(* IEC 61131-3 sources: repolevel_ST_code_completion/output/full_case_fixed/repoeval_elevator/readful_result, 5 files *)

(* ---- F_DetectCurrentFloor.st ---- *)
FUNCTION F_DetectCurrentFloor : INT
VAR_INPUT
FloorSensor0	:	BOOL;		// 0楼传感器
FloorSensor1	:	BOOL;		// 1楼传感器
FloorSensor2	:	BOOL;		// 2楼传感器
FloorSensor3	:	BOOL;		// 3楼传感器
CurrentFloor	:	INT;		// 当前楼层（用于保持状态）
END_VAR
IF FloorSensor0 THEN
F_DetectCurrentFloor := 0;
ELSIF FloorSensor1 THEN
F_DetectCurrentFloor := 1;
ELSIF FloorSensor2 THEN
F_DetectCurrentFloor := 2;
ELSIF FloorSensor3 THEN
F_DetectCurrentFloor := 3;
ELSE
F_DetectCurrentFloor := 0; // Default valid floor value if no sensors are active
END_IF;
RETURN;
END_FUNCTION

(* ---- F_RegisterCalls.st ---- *)
FUNCTION F_RegisterCalls
VAR_INPUT
 CallGround		:	BOOL;		// 0楼呼叫
 CallFloor1		:	BOOL;		// 1楼呼叫
 CallFloor2		:	BOOL;		// 2楼呼叫
 CallFloor3		:	BOOL;		// 3楼呼叫
END_VAR
VAR_IN_OUT
 TargetFloors	:	ARRAY[0..3] OF BOOL;	// 目标楼层数组
END_VAR
IF CallGround THEN
 TargetFloors[0] := TRUE;
END_IF

IF CallFloor1 THEN
 TargetFloors[1] := TRUE;
END_IF

IF CallFloor2 THEN
 TargetFloors[2] := TRUE;
END_IF

IF CallFloor3 THEN
 TargetFloors[3] := TRUE;
END_IF

RETURN;
END_FUNCTION

(* ---- F_UpdateDoorAnimation.st ---- *)
FUNCTION F_UpdateDoorAnimation : DINT
VAR_INPUT
bOpenDoor		:	BOOL;		// 开门命令
bCloseDoor		:	BOOL;		// 关门命令
bCallFloor		:	BOOL;		// 该楼层有呼叫
nCurrentAni		:	DINT;		// 当前动画值
nMaxAni			:	DINT := 70;	// 最大动画值
END_VAR
VAR
nNewAni			:	DINT;		// 新的动画值
END_VAR

nNewAni := nCurrentAni;

// 开门动画（增加动画值）
IF bOpenDoor AND nNewAni < nMaxAni AND bCallFloor THEN
nNewAni := nNewAni + 1;
END_IF

// 关门动画（减少动画值）
IF bCloseDoor AND nNewAni > 0 THEN
nNewAni := nNewAni - 1;
END_IF

F_UpdateDoorAnimation := nNewAni;
END_FUNCTION

(* ---- FB_ElevatorDoorController.st ---- *)
FUNCTION_BLOCK FB_ElevatorDoorController
VAR_INPUT
	bArrivedAtTarget	:	BOOL;		// 到达目标楼层
	bDoorClosed			:	BOOL;		// 门已关闭传感器
END_VAR
VAR_OUTPUT
	bOpenDoor			:	BOOL;		// 开门命令
	bCloseDoor			:	BOOL;		// 关门命令
	bDoorOpen			:	BOOL;		// 门打开状态
	bDoorReady			:	BOOL;		// 门准备好（可以移动）
END_VAR
VAR
	fbDoorTimer			:	TON;		// 开门延时定时器
	fbCloseDoorTimer	:	TON;		// 关门延时定时器
	nState				:	INT;		// 状态机
END_VAR

CASE nState OF
	0: // 空闲状态
		bOpenDoor := FALSE;
		bCloseDoor := FALSE;
		bDoorReady := TRUE;

		IF bArrivedAtTarget THEN
			nState := 1; // 开始开门流程
		END_IF

1: // 开门延时
    bCloseDoor := FALSE;
    bDoorReady := FALSE;
    fbDoorTimer.IN := TRUE;
    fbDoorTimer.PT := T#2S;

    IF fbDoorTimer.Q THEN
      fbDoorTimer.IN := FALSE;
      nState := 2; // 开门命令
    END_IF

	2: // 开门命令
		bOpenDoor := TRUE;
		bDoorOpen := TRUE;
		bDoorReady := FALSE;

		IF NOT bArrivedAtTarget THEN
			nState := 3; // 开始关门流程
		END_IF

3: // 关门延时
    bOpenDoor := FALSE;
    bDoorReady := FALSE;
    fbCloseDoorTimer.IN := TRUE;
    fbCloseDoorTimer.PT := T#2S;

    IF fbCloseDoorTimer.Q THEN
      fbCloseDoorTimer.IN := FALSE;
      nState := 4; // 关门命令
    END_IF

	4: // 关门命令
		bCloseDoor := TRUE;
		bDoorOpen := FALSE;

		IF bDoorClosed THEN
			bCloseDoor := FALSE;
			bDoorReady := TRUE;
			nState := 0; // 返回空闲状态
		END_IF

# Removed this segment as Structured Text does not support ELSE for CASE statements.
# The default case is already handled as RETURNS to 'nState := 0'.
END_CASE
END_FUNCTION_BLOCK

(* ---- FB_ElevatorMovement.st ---- *)
FUNCTION_BLOCK FB_ElevatorMovement
VAR_INPUT
	CurrentFloor		:	INT;				// 当前楼层
	bDoorReady			:	BOOL;				// 门准备好
END_VAR
VAR_IN_OUT
	TargetFloors		:	ARRAY[0..3] OF BOOL;	// 目标楼层数组
END_VAR
VAR_OUTPUT
	bMovingUp			:	BOOL;				// 向上移动
	bMovingDown			:	BOOL;				// 向下移动
	bArrivedAtTarget	:	BOOL;				// 到达目标楼层
END_VAR
VAR
	fbMoveDelayTimer	:	TON;				// 移动延时定时器
	i					:	INT;				// 循环变量
	bHasUpperRequest	:	BOOL;				// 有更高楼层请求
	bHasLowerRequest	:	BOOL;				// 有更低楼层请求
END_VAR

// 检查是否到达目标楼层
IF (CurrentFloor >= 0) AND (CurrentFloor <= 3) THEN // 添加边界检查以避免数组越界
  IF TargetFloors[CurrentFloor] THEN
    bArrivedAtTarget := TRUE;
    TargetFloors[CurrentFloor] := FALSE; // 清除请求
    bMovingUp := FALSE;
    bMovingDown := FALSE;
  ELSE
    bArrivedAtTarget := FALSE;
  END_IF
END_IF

// 检查是否有更高或更低楼层的请求
bHasUpperRequest := FALSE;
bHasLowerRequest := FALSE;

FOR i := 0 TO 3 DO
  IF TargetFloors[i] THEN
   IF i > CurrentFloor THEN
    bHasUpperRequest := TRUE;
   ELSIF i < CurrentFloor THEN
    bHasLowerRequest := TRUE;
   END_IF
  END_IF
END_FOR

// 控制电梯移动方向
IF bDoorReady THEN
	IF bHasUpperRequest AND NOT bHasLowerRequest THEN
		bMovingUp := TRUE;
		bMovingDown := FALSE;
	ELSIF bHasLowerRequest AND NOT bHasUpperRequest THEN
		bMovingUp := FALSE;
		bMovingDown := TRUE;
	ELSIF bHasUpperRequest AND bHasLowerRequest THEN
		IF bMovingUp THEN
			// 如果当前向上移动，继续向上移动
			bMovingUp := TRUE;
			bMovingDown := FALSE;
		ELSIF bMovingDown THEN
			// 如果当前向下移动，继续向下移动
			bMovingUp := FALSE;
			bMovingDown := TRUE;
		END_IF
	ELSE
		// 没有请求时停止移动
		bMovingUp := FALSE;
		bMovingDown := FALSE;
	END_IF
END_IF
END_FUNCTION_BLOCK
